FUNCTION_BLOCK Piper_EM EXTENDS PiperModule
VAR_INPUT
END_VAR
VAR_OUTPUT
END_VAR
VAR
    task : REFERENCE TO TaskFB;
    keepExecuting : BOOL := TRUE;
END_VAR

// Copyright (c) 2024 Loupe (https://loupe.team), provided under the MIT License.

METHOD Executing : MACHINE_STATE
// Copyright (c) 2024 Loupe (https://loupe.team), provided under the MIT License.

WHILE keepExecuting DO
    ;
    //
END_WHILE
END_METHOD

METHOD FB_init : BOOL
VAR_INPUT
    bInitRetains : BOOL; // if TRUE, the retain variables are initialized (warm start / cold start)
    bInCopyCode : BOOL; // if TRUE, the instance afterwards gets moved into the copy code (online change)
    machineIn : REFERENCE TO Piper;
    taskFB : REFERENCE TO TaskFB;
    //	context : IPluginRunner;
END_VAR
// Copyright (c) 2024 Loupe (https://loupe.team), provided under the MIT License.

THIS^.setContext(taskFB);
task REF= taskFB;
END_METHOD

END_FUNCTION_BLOCK

(* stored: Version 1.1.0.1
   POU Piper_EM: Id {f5bdbed5-22e7-4707-a8a6-280efebba65a}, SpecialFunc None
   Method Executing: Id {687a8988-295f-0d32-36fb-3c36085d63e6}
   Method FB_init: Id {849118c9-b30c-4253-9dc8-45fb450e8398} *)
